// TIA Portal V20 export
DATA_BLOCK "Pallets_Stations"   // DB11
{ S7_Optimized_Access := 'TRUE' }
// stored: MemoryReserve 100
   VAR RETAIN
      Pallets : Array[1..24] of "Pallet";
   END_VAR
   VAR
      Stations : Array[1..4, 1..12] of "Station";
      Stations_ROW1 : Array[1..12] of "StationLight";
      Stations_ROW2 { S7_SetPoint := 'True'} : Array[1..12] of "StationLight";
      Stations_ROW3 { S7_SetPoint := 'True'} : Array[1..12] of "StationLight";
      Stations_ROW4 { S7_SetPoint := 'True'} : Array[1..12] of "StationLight";
   END_VAR
BEGIN
   Stations[1,1..12].Numer := 1;
   Stations[2,1..12].Numer := 2;
   Stations[3,1..12].Numer := 3;
   Stations[4,1..12].Numer := 4;
   Stations[1,1..12].Row := 1;
   Stations[2,1..12].Row := 2;
   Stations[3,1..12].Row := 3;
   Stations[4,1..12].Row := 4;
   Stations[1,1].Column := 1;
   Stations[1,2].Column := 2;
   Stations[1,3].Column := 3;
   Stations[1,4].Column := 4;
   Stations[1,5].Column := 5;
   Stations[1,6].Column := 6;
   Stations[1,7].Column := 7;
   Stations[1,8].Column := 8;
   Stations[1,9].Column := 9;
   Stations[1,10].Column := 10;
   Stations[1,11].Column := 11;
   Stations[1,12].Column := 12;
   Stations[2,1].Column := 1;
   Stations[2,2].Column := 2;
   Stations[2,3].Column := 3;
   Stations[2,4].Column := 4;
   Stations[2,5].Column := 5;
   Stations[2,6].Column := 6;
   Stations[2,7].Column := 7;
   Stations[2,8].Column := 8;
   Stations[2,9].Column := 9;
   Stations[2,10].Column := 10;
   Stations[2,11].Column := 11;
   Stations[2,12].Column := 12;
   Stations[3,1].Column := 1;
   Stations[3,2].Column := 2;
   Stations[3,3].Column := 3;
   Stations[3,4].Column := 4;
   Stations[3,5].Column := 5;
   Stations[3,6].Column := 6;
   Stations[3,7].Column := 7;
   Stations[3,8].Column := 8;
   Stations[3,9].Column := 9;
   Stations[3,10].Column := 10;
   Stations[3,11].Column := 11;
   Stations[3,12].Column := 12;
   Stations[4,1].Column := 1;
   Stations[4,2].Column := 2;
   Stations[4,3].Column := 3;
   Stations[4,4].Column := 4;
   Stations[4,5].Column := 5;
   Stations[4,6].Column := 6;
   Stations[4,7].Column := 7;
   Stations[4,8].Column := 8;
   Stations[4,9].Column := 9;
   Stations[4,10].Column := 10;
   Stations[4,11].Column := 11;
   Stations[4,12].Column := 12;
   Stations_ROW1[1].Numer := 35;
   Stations_ROW1[2].Numer := 34;
   Stations_ROW1[3].Numer := 33;
   Stations_ROW1[4].Numer := 32;
   Stations_ROW1[5].Numer := 31;
   Stations_ROW1[6].Numer := 30;
   Stations_ROW1[7].Numer := 29;
   Stations_ROW1[8].Numer := 28;
   Stations_ROW1[9].Numer := 27;
   Stations_ROW1[10].Numer := 26;
   Stations_ROW1[11].Numer := 25;
   Stations_ROW2[1].Numer := 02;
   Stations_ROW2[2].Numer := 1;
   Stations_ROW2[3].Numer := 38;
   Stations_ROW2[4].Numer := 36;
   Stations_ROW2[5].Numer := 37;
   Stations_ROW2[6].Numer := 18;
   Stations_ROW2[7].Numer := 19;
   Stations_ROW2[8].Numer := 20;
   Stations_ROW2[9].Numer := 21;
   Stations_ROW2[10].Numer := 22;
   Stations_ROW2[11].Numer := 23;
   Stations_ROW2[12].Numer := 24;
   Stations_ROW3[1].Numer := 3;
   Stations_ROW3[11].Numer := 17;
   Stations_ROW4[1].Numer := 4;
   Stations_ROW4[2].Numer := 5;
   Stations_ROW4[3].Numer := 6;
   Stations_ROW4[4].Numer := 7;
   Stations_ROW4[5].Numer := 8;
   Stations_ROW4[6].Numer := 9;
   Stations_ROW4[7].Numer := 10;
   Stations_ROW4[8].Numer := 11;
   Stations_ROW4[9].Numer := 12;
   Stations_ROW4[10].Numer := 13;
   Stations_ROW4[11].Numer := 14;
END_DATA_BLOCK
